FUNCTION_BLOCK FlashSignal
VAR_INPUT
  flash_time: TIME;
END_VAR
VAR_OUTPUT
	q: BOOL;
END_VAR
VAR
	timer_flash: TON;
END_VAR

timer_flash(IN:=TRUE, PT:=flash_time);
IF (timer_flash.Q) THEN
	timer_flash(IN:=FALSE);
	q := NOT q;
END_IF

METHOD FB_init : BOOL
VAR_INPUT
	bInitRetains : BOOL; // if TRUE, the retain variables are initialized (warm start / cold start)
	bInCopyCode : BOOL;  // if TRUE, the instance afterwards gets moved into the copy code (online change)
  flash_time: TIME;
END_VAR
THIS^.flash_time := flash_time;
END_METHOD

END_FUNCTION_BLOCK

(* stored: Version 1.1.0.1, ProductVersion 3.1.4022.18
   POU FlashSignal: Id {c3ea18fd-76fb-4f8e-b352-e9455e19b9e8}, SpecialFunc None
   Method FB_init: Id {f3ff670d-7fe2-45dc-bc8a-ba58920184f9} *)
